//{attribute 'qualified_only'}
{attribute 'strict'}
TYPE E_StateMachine :
(
	eOff	 := 0,
	eOn  	 := 1,
	eForward := 2,
	eReverse := 3,
	eFault   := 4,
	eAuto    := 5
		
);
END_TYPE

(* stored: Version 1.1.0.1, ProductVersion 3.1.4024.12
   EnumerationTextList E_StateMachine: Id {fee97b33-5cc6-4b0a-b875-59cb7cf6c183} *)
